// TwinCAT 3 PLC project PLCPROJECT
// ProgramVersion: 3.1.4024.0
// libraries:
//   Tc2_Standard, * (Beckhoff Automation GmbH)
//   Tc2_System, * (Beckhoff Automation GmbH)
//   Tc3_Module, * (Beckhoff Automation GmbH)
// project tree:
//   / PlcTask.TcTTO
//   POUs/ Light.TcPOU, MAIN.TcPOU
// real-time tasks:
//   TASK PlcTask: cycle T#10ms, priority 20, ADS port 350

CONFIGURATION PLCPROJECT
    RESOURCE PLC ON TwinCAT3
        TASK PlcTask(INTERVAL := T#10ms, PRIORITY := 20);
        PROGRAM MAIN WITH PlcTask : MAIN;
    END_RESOURCE
END_CONFIGURATION

// ---- POUs/MAIN.TcPOU
PROGRAM MAIN
VAR
	output1: BOOL;
	input1 : BOOL;
	andrew : DWORD;
	counter : Int;
END_VAR

counter := counter +1;

END_PROGRAM

// ---- POUs/Light.TcPOU
PROGRAM Light
VAR
	Lamp : BOOL;
END_VAR

END_PROGRAM
